(*
SPDX-FileCopyrightText: © 2026 Oleksandr Tiutyk <trofimich@gmail.com>
SPDX-License-Identifier: MIT
License: https://opensource.org/license/mit
*)

INTERFACE IGenericConversionNotSupportedException EXTENDS IGeneralException

METHOD Throw
VAR_INPUT
	sourceNamespaceName : STRING;
	sourceClassName : STRING;
	sourcePOUName : STRING;
	sourcePosition : STRING;
	sourceDataType : GENERIC_TYPE_CLASS;
	targetDataType : GENERIC_TYPE_CLASS;
END_VAR
END_METHOD

END_INTERFACE

(* stored: Version 1.1.0.1
   Itf IGenericConversionNotSupportedException: Id {67a2a108-d3bc-4b19-a1e1-b16c2025427d}
   Method Throw: Id {4d375bbc-f9a2-4054-a53e-6b0ca0ca138f} *)
